FUNCTION_BLOCK POU_NCPowerOn
VAR_INPUT
END_VAR
VAR_OUTPUT
END_VAR
VAR
	XAxisPowerOn: MC_Power;
	GoMotor: MC_MoveVelocity;
	direction: MC_Direction;
	TRUEB: BOOL;
	MoveDistance: MC_MoveModulo;
	MoveBack: MC_MoveModulo;
	DoneT: BOOL;
END_VAR

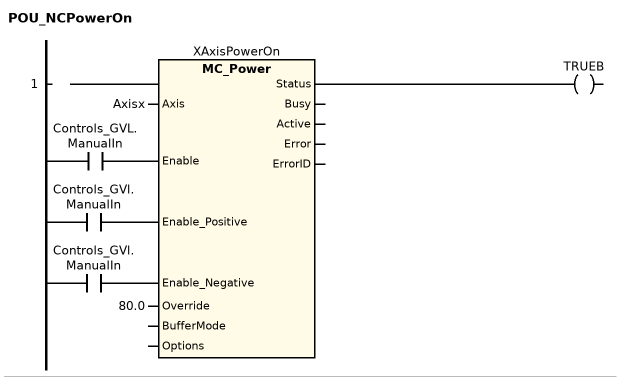
// NETWORK 1
XAxisPowerOn(
    Axis := Axisx,
    Enable := Controls_GVL.ManualIn,
    Enable_Positive := Controls_GVl.ManualIn,
    Enable_Negative := Controls_GVl.ManualIn,
    Override := 80.0); // MC_Power
TRUEB := XAxisPowerOn.Status;

END_FUNCTION_BLOCK

(* stored: Version 1.1.0.1, ProductVersion 3.1.4024.2
   POU POU_NCPowerOn: Id {4a36d793-c8a0-4f4b-8dbf-c4d29d54fc48}, SpecialFunc None *)
